// TIA Portal V20 export
TYPE "LCFL_typeMTPOSLevel"
TITLE = MTP for OS level / MTP für OS-Level
// MTP data for OS level / MTP-Daten für OS-Level
   STRUCT
      OSLevel : Byte := 16#00;   // OS-Level / OS level
   END_STRUCT;
END_TYPE
